// TwinCAT 3 PLC project PlcIotHttpSampleMindsphere
// ProgramVersion: 3.1.4023.0
// libraries:
//   Tc2_Standard, * (Beckhoff Automation GmbH)
//   Tc2_System, * (Beckhoff Automation GmbH)
//   Tc3_IotBase, * (Beckhoff Automation GmbH)
//   Tc3_Module, * (Beckhoff Automation GmbH)
// project tree:
//   / PlcTask.TcTTO
//   POUs/ MAIN.TcPOU
//   POUs/Mindsphere/ FB_TestHTTP_Mindsphere_AcquireAAT.TcPOU, FB_TestHTTP_Mindsphere_CreateDataSource.TcPOU, FB_TestHTTP_Mindsphere_CreateMapping.TcPOU, FB_TestHTTP_Mindsphere_GetDataSource.TcPOU, FB_TestHTTP_Mindsphere_KeyRotation.TcPOU, FB_TestHTTP_Mindsphere_Onboarding.TcPOU
// real-time tasks:
//   TASK PlcTask: cycle T#10ms, priority 20, ADS port 350

CONFIGURATION PlcIotHttpSampleMindsphere
    RESOURCE PLC ON TwinCAT3
        TASK PlcTask(INTERVAL := T#10ms, PRIORITY := 20);
        PROGRAM MAIN WITH PlcTask : MAIN;
    END_RESOURCE
END_CONFIGURATION

// ---- POUs/MAIN.TcPOU
PROGRAM MAIN
VAR
	// trigger command execution for Siemens Mindsphere samples
	bOnboardMindsphere				: BOOL;
	bKeyRotationMindsphere			: BOOL;
	bAcquireAATMindsphere			: BOOL;
	bCreateDataSourceMindsphere		: BOOL;
	bGetDataSourceMindsphere		: BOOL;
	bCreateMappingMindsphere		: BOOL;
	
	fbHttpClientMindsphere			: FB_IotHttpClient :=(sHostName:='gateway.eu1.mindsphere.io',
									bKeepAlive:=TRUE, tConnectionTimeout:=T#10S);						
	
	fbHttpMindsphereOnboarding		: FB_TestHTTP_Mindsphere_Onboarding;
	fbHttpMindsphereKeyRotation		: FB_TestHTTP_Mindsphere_KeyRotation;
	fbHttpMindsphereAcquireAAT		: FB_TestHTTP_Mindsphere_AcquireAAT;
	fbHttpMindsphereCreateDataSource: FB_TestHTTP_Mindsphere_CreateDataSource;
	fbHttpMindsphereGetDataSource	: FB_TestHTTP_Mindsphere_GetDataSource;
	fbHttpMindsphereCreateMapping	: FB_TestHTTP_Mindsphere_CreateMapping;
END_VAR

// init client parameters at startup
IF NOT fbHttpClientMindsphere.bConfigured THEN 
	fbHttpClientMindsphere.stTLS.sCA:= 'C:\TwinCAT\3.1\Config\Certificates\Mindsphere\MindsphereRoot_Europe.pem';
	fbHttpClientMindsphere.nHostPort:= 443;
	fbHttpClientMindsphere.stTLS.bNoServerCertCheck:= TRUE;
END_IF

IF fbHttpClientMindsphere.bConfigured THEN
 	fbHttpMindsphereOnboarding(bSend:=bOnboardMindsphere, fbClient:=fbHttpClientMindsphere);
	fbHttpMindsphereKeyRotation(bSend:=bKeyRotationMindsphere, fbClient:=fbHttpClientMindsphere);
	fbHttpMindsphereAcquireAAT(bSend:=bAcquireAATMindsphere, fbClient:=fbHttpClientMindsphere);
	fbHttpMindsphereCreateDataSource(bSend:=bCreateDataSourceMindsphere, fbClient:=fbHttpClientMindsphere);
	fbHttpMindsphereGetDataSource(bSend:=bGetDataSourceMindsphere, fbClient:=fbHttpClientMindsphere);
	fbHttpMindsphereCreateMapping(bSend:=bCreateMappingMindsphere, fbClient:=fbHttpClientMindsphere);
END_IF

fbHttpClientMindsphere.Execute();

END_PROGRAM

// ---- POUs/Mindsphere/FB_TestHTTP_Mindsphere_Onboarding.TcPOU
FUNCTION_BLOCK FB_TestHTTP_Mindsphere_Onboarding
VAR_INPUT
	bSend				: BOOL;
END_VAR
VAR_IN_OUT
	fbClient			: FB_IotHttpClient;
END_VAR
VAR_OUTPUT
	bBusy				: BOOL;
	bError				: BOOL;
END_VAR
VAR	
	fbRequest			: FB_IotHttpRequest;
	fbHeader			: FB_IotHttpHeaderFieldMap;
	fbJson				: FB_JsonDomParser;
	nState				: UDINT;
	RisingEdge			: R_TRIG;
	
	bGetContentResult	: BOOL;
	sContent			: STRING(2048);
	
	bGetJsonResult		: BOOL;
	jsonDoc				: SJsonValue;
	jsonVal				: SJsonValue;
	sResultValue		: STRING;
	
	nReqCount			: UDINT;
	nResCount			: UDINT;
	nValidResCount		: UDINT;
	nErrCount			: UDINT;	
END_VAR

RisingEdge(CLK:= bSend);
CASE nState OF
0:		
	IF RisingEdge.Q THEN
		sContent := '{}';
		fbHeader.AddField('Content-Type', 'application/json', FALSE);
		fbHeader.AddField('Authorization', 'Bearer eyJraWQiOiJrZXktaWQtMSIsInR5cCI6IkpXVCIsImFsZyI6IlJTMjU2In0.eyJpc3MiOiJTQ0kiLCJzdWIiOiI5NTZjY2UzNjA1YjE0MjA4OTAwOTVlNTBlMmIxMWUxNyIsImF1ZCI6IkFJQU0iLCJpYXQiOjE1ODIxODUxMzMsIm5iZiI6MTU4MjE4NTEzMywiZXhwIjoxNTgyNzg5OTMzLCJqdGkiOiIxYWI0Y2U4MS1jOWJhLTQ2MzctYjIyNy0xYmZjNjk5MWI4NGEiLCJzY29wZSI6IklBVCIsInRlbiI6ImJlY2tob2ZmIiwidGVuX2N0eCI6Im1haW4tdGVuYW50IiwiY2xpZW50X2NyZWRlbnRpYWxzX3Byb2ZpbGUiOlsiU0hBUkVEX1NFQ1JFVCJdLCJzY2hlbWFzIjpbInVybjpzaWVtZW5zOm1pbmRzcGhlcmU6djEiXX0.mOtfZ4WU-8C8r2SggtAEXPS6e1dGlTl4IhrB8WwrWN-FoJE5Tq1DR5j2pSnBRtEuBcrJhd3_Lu2kQ_YdJxJwrPnw_7XdTjqc-LavqDZUUZhOQGqVCurarsKkKcYUMGC8WDLXG81z64l4vrjYSC6drq7ZXVYZVWa-MyHQSWoxQ9QJv1hy_dNYjL6mNf6rmlSqhbzQGo3-3_y5pb7AptIPwYB7GHeH5Iw28PJxjjrWP18ifQlDZYz4AmLGYzdyvGWbbAeHjrdkI8GXls7yhBZ_xIcFwYT72UsDaxG_SIA5YqWhBCyyNM-ElInfPW2PAwe3irzbxinKO3uhstYjJqN3Rg', FALSE);
		IF fbRequest.SendRequest(sUri:= '/api/agentmanagement/v3/register', fbClient:= fbClient, eRequestType:= ETcIotHttpRequestType.HTTP_POST, pContent:= ADR(sContent), nContentSize:= LEN2(ADR(sContent)), fbHeader:= fbHeader) THEN				
			nState:= 1;
			nReqCount:= nReqCount+1;
			bBusy:= TRUE;
			bError:= FALSE;
		END_IF					
	END_IF
1:
	IF NOT fbRequest.bBusy THEN
		bError:= TRUE;
		IF NOT fbRequest.bError THEN				 				
			bGetContentResult:= fbRequest.GetContent(pContent:= ADR(sContent), nContentSize:= SIZEOF(sContent), bSetNullTermination:= TRUE);	
			IF fbRequest.nStatusCode >= 200 AND fbRequest.nStatusCode < 300 THEN
				bGetJsonResult:= FALSE;
				jsonDoc:= fbRequest.GetJsonDomContent(fbJson);				
				(* Parse Onboarding response in order to acquire:
					client_id
					client_secret
					client_secret_expires_at
					regsitration_access_token (RAT)
					registration_client_uri 
				*)
				nResCount:= nResCount+1;					
			END_IF				
		END_IF
		nState:= 0;
		bBusy:= FALSE;
		IF bError THEN
			nErrCount:= nErrCount+1;
		END_IF		
	END_IF  	
END_CASE

END_FUNCTION_BLOCK

// ---- POUs/Mindsphere/FB_TestHTTP_Mindsphere_KeyRotation.TcPOU
FUNCTION_BLOCK FB_TestHTTP_Mindsphere_KeyRotation
VAR_INPUT
	bSend				: BOOL;
END_VAR
VAR_IN_OUT
	fbClient			: FB_IotHttpClient;
END_VAR
VAR_OUTPUT
	bBusy				: BOOL;
	bError				: BOOL;
END_VAR
VAR	
	fbRequest			: FB_IotHttpRequest;
	fbHeader			: FB_IotHttpHeaderFieldMap;
	fbJson				: FB_JsonDomParser;
	nState				: UDINT;
	RisingEdge			: R_TRIG;
	
	bGetContentResult	: BOOL;
	sContent			: STRING(2048);
	
	bGetJsonResult		: BOOL;
	jsonDoc				: SJsonValue;
	jsonVal				: SJsonValue;
	sResultValue		: STRING;
	
	nReqCount			: UDINT;
	nResCount			: UDINT;
	nValidResCount		: UDINT;
	nErrCount			: UDINT;	
END_VAR

RisingEdge(CLK:= bSend);
CASE nState OF
0:		
	IF RisingEdge.Q THEN
		sContent := '{ "client_id": "956cce3605b1420890095e50e2b11e17" }';
		fbHeader.AddField('Content-Type', 'application/json', FALSE);
		// Header field 'Authorization' now includes RAT 
		fbHeader.AddField('Authorization', 'Bearer eyJraWQiOiJrZXktaWQtMSIsInR5cCI6IkpXVCIsImFsZyI6IlJTMjU2In0.eyJpc3MiOiJTQ0kiLCJzdWIiOiI5NTZjY2UzNjA1YjE0MjA4OTAwOTVlNTBlMmIxMWUxNyIsImF1ZCI6IkFJQU0iLCJpYXQiOjE1ODIxODcwNTEsIm5iZiI6MTU4MjE4NzA1MSwiZXhwIjozMTU1Njg4OTg2NDQwMzE5OSwianRpIjoiNzYzM2ViZjctNWY1ZS00NWI3LTkwOTctYzEyODRkZWU2ZjNjIiwic2NvcGUiOiJSQVQiLCJ0ZW4iOiJiZWNraG9mZiIsInRlbl9jdHgiOiJtYWluLXRlbmFudCIsImNsaWVudF9jcmVkZW50aWFsc19wcm9maWxlIjpbIlNIQVJFRF9TRUNSRVQiXSwic2NoZW1hcyI6WyJ1cm46c2llbWVuczptaW5kc3BoZXJlOnYxIl19.dE3IGrI0JIY6O6nYmLp0F3yxHYIvTzQtT9d7ZL7X5MdKMXUeO6G_nXl2MFgEnThPm400hqtsOkLUO1MptoFFlg3rOj227p2--hYN4zLIefDKd54tG0dZ0K7HuX7_oMBjRKoUzF6ls7ujfGyjYH4o0A3FW42mZCecmZxLJmcYoWi7J5iF6oLMZc--Yg1O5RTXwkjp0pwRNMJVS_xofNAdPxg3wvIYjsraUl_TGLPswG_JnsNuYhnRtGfrG23zg1IlSszkB-RYwnzLvsep6ACAfVRlsJve0CN6zU87W0GboH7s_aDAAVTlxbNMz3Tvu44gOk0FmhDoMOvb20peNyg9Iw', FALSE);
		IF fbRequest.SendRequest(sUri:= '/api/agentmanagement/v3/register/956cce3605b1420890095e50e2b11e17', fbClient:= fbClient, eRequestType:= ETcIotHttpRequestType.HTTP_PUT, pContent:= ADR(sContent), nContentSize:= LEN2(ADR(sContent)), fbHeader:= fbHeader) THEN				
			nState:= 1;
			nReqCount:= nReqCount+1;
			bBusy:= TRUE;
			bError:= FALSE;
		END_IF					
	END_IF
1:
	IF NOT fbRequest.bBusy THEN
		bError:= TRUE;
		IF NOT fbRequest.bError THEN				 				
			bGetContentResult:= fbRequest.GetContent(pContent:= ADR(sContent), nContentSize:= SIZEOF(sContent), bSetNullTermination:= TRUE);	
			IF fbRequest.nStatusCode >= 200 AND fbRequest.nStatusCode < 300 THEN
				bGetJsonResult:= FALSE;
				jsonDoc:= fbRequest.GetJsonDomContent(fbJson);				
				(* Parse KeyRotation response in order to acquire:
					client_id
					client_secret
					client_secret_expires_at
					regsitration_access_token (RAT)
					registration_client_uri 
				*)
				nResCount:= nResCount+1;					
			END_IF				
		END_IF
		nState:= 0;
		bBusy:= FALSE;
		IF bError THEN
			nErrCount:= nErrCount+1;
		END_IF		
	END_IF  	
END_CASE

END_FUNCTION_BLOCK

// ---- POUs/Mindsphere/FB_TestHTTP_Mindsphere_AcquireAAT.TcPOU
FUNCTION_BLOCK FB_TestHTTP_Mindsphere_AcquireAAT
VAR_INPUT
	bSend				: BOOL;
END_VAR
VAR_IN_OUT
	fbClient			: FB_IotHttpClient;
END_VAR
VAR_OUTPUT
	bBusy				: BOOL;
	bError				: BOOL;
END_VAR
VAR	
	fbRequest			: FB_IotHttpRequest;
	fbHeader			: FB_IotHttpHeaderFieldMap;
	fbJson				: FB_JsonDomParser;
	nState				: UDINT;
	RisingEdge			: R_TRIG;
	
	bGetContentResult	: BOOL;
	sContent			: STRING(2048);
	
	bGetJsonResult		: BOOL;
	jsonDoc				: SJsonValue;
	jsonVal				: SJsonValue;
	sResultValue		: STRING;
	
	nReqCount			: UDINT;
	nResCount			: UDINT;
	nValidResCount		: UDINT;
	nErrCount			: UDINT;	
END_VAR

RisingEdge(CLK:= bSend);
CASE nState OF
0:		
	IF RisingEdge.Q THEN
		sContent := 'grant_type=client_credentials&client_assertion_type=urn:ietf:params:oauth:client-assertion-type:jwt-bearer&client_assertion=eyJ0eXAiOiJKV1QiLCJhbGciOiJIUzI1NiJ9.eyJpc3MiOiI5NTZjY2UzNjA1YjE0MjA4OTAwOTVlNTBlMmIxMWUxNyIsInN1YiI6Ijk1NmNjZTM2MDViMTQyMDg5MDA5NWU1MGUyYjExZTE3IiwiYXVkIjpbInNvdXRoZ2F0ZSJdLCJpYXQiOjE1ODIxOTI2NjEsIm5iZiI6MTU4MjE5MjY2MSwiZXhwIjoxNTgyMTkzNjYxLCJqdGkiOiJjNDJlYjNiYy04NjI2LTQ3ZDktOTRjYy01MWE0OGQ3ZTc3YjMiLCJ0ZW4iOiJiZWNraG9mZiIsInNjaGVtYXMiOlsidXJuOnNpZW1lbnM6bWluZHNwaGVyZTp2MSJdfQ.LZcYDd38oRX1rdwGeBuqJVy5S4ja4Bmo5lvTW-EloP4';
		fbHeader.AddField('Content-Type', 'application/x-www-form-urlencoded', FALSE);
		IF fbRequest.SendRequest(sUri:= '/api/agentmanagement/v3/oauth/token', fbClient:= fbClient, eRequestType:= ETcIotHttpRequestType.HTTP_POST, pContent:= ADR(sContent), nContentSize:= LEN2(ADR(sContent)), fbHeader:= fbHeader) THEN				
			nState:= 1;
			nReqCount:= nReqCount+1;
			bBusy:= TRUE;
			bError:= FALSE;
		END_IF					
	END_IF
1:
	IF NOT fbRequest.bBusy THEN
		bError:= TRUE;
		IF NOT fbRequest.bError THEN				 				
			bGetContentResult:= fbRequest.GetContent(pContent:= ADR(sContent), nContentSize:= SIZEOF(sContent), bSetNullTermination:= TRUE);	
			IF fbRequest.nStatusCode >= 200 AND fbRequest.nStatusCode < 300 THEN
				bGetJsonResult:= FALSE;
				jsonDoc:= fbRequest.GetJsonDomContent(fbJson);				
				(* Parse AAT API Call response in order to acquire:
					access_token
					token_type
					expires_in
					scope
					jti 
				*)
				nResCount:= nResCount+1;					
			END_IF				
		END_IF
		nState:= 0;
		bBusy:= FALSE;
		IF bError THEN
			nErrCount:= nErrCount+1;
		END_IF		
	END_IF  	
END_CASE

END_FUNCTION_BLOCK

// ---- POUs/Mindsphere/FB_TestHTTP_Mindsphere_CreateDataSource.TcPOU
FUNCTION_BLOCK FB_TestHTTP_Mindsphere_CreateDataSource
VAR_INPUT
	bSend				: BOOL;
END_VAR
VAR_IN_OUT
	fbClient			: FB_IotHttpClient;
END_VAR
VAR_OUTPUT
	bBusy				: BOOL;
	bError				: BOOL;
END_VAR
VAR	
	fbRequest			: FB_IotHttpRequest;
	fbHeader			: FB_IotHttpHeaderFieldMap;
	fbJson				: FB_JsonDomParser;
	nState				: UDINT;
	RisingEdge			: R_TRIG;
	
	bGetContentResult	: BOOL;
	sContent			: STRING(2048);
	
	bGetJsonResult		: BOOL;
	jsonDoc				: SJsonValue;
	jsonVal				: SJsonValue;
	sResultValue		: STRING;
	
	nReqCount			: UDINT;
	nResCount			: UDINT;
	nValidResCount		: UDINT;
	nErrCount			: UDINT;	
END_VAR

RisingEdge(CLK:= bSend);
CASE nState OF
0:		
	IF RisingEdge.Q THEN
		// Body includes JSON document with DataSource configuration that should be created
		sContent := '{"configurationId":"Device_DataSource","dataSources":[{"name":"Device_DataSource_Data","customData":null,"description":"","dataPoints":[{"id":"PWR_OUT","name":"PWR_OUT","description":"","unit":"MW","type":"DOUBLE","customData":null},{"id":"V_OUT","name":"V_OUT","description":"","unit":"Volt","type":"DOUBLE","customData":null}]}]}';
		fbHeader.AddField('Content-Type', 'application/json', FALSE);
		fbHeader.AddField('If-Match', '0', FALSE);
		// Header field 'Authorization' now includes AAT 
		fbHeader.AddField('Authorization', 'Bearer eyJraWQiOiJrZXktaWQtMSIsImFsZyI6IlJTMjU2IiwidHlwIjoiSldUIn0.eyJqdGkiOiJjNzgzOTg1OC1mYmQ4LTQ5YTQtOTE5Yy03YjFmN2FiMDQ3ZjUiLCJzY29wZSI6WyJtZHNwOmNvcmU6RGVmYXVsdEFnZW50Il0sImlzcyI6Imh0dHBzOi8vc291dGhnYXRlLmV1MS5taW5kc3BoZXJlLmlvL2FwaS9hZ2VudG1hbmFnZW1lbnQvIiwic3ViIjoiZTFmODRkM2VkMGIzNDljY2JjYWQxZTkwMzgxMzE5ZTIiLCJ6aWQiOiJhZ2VudGlhbSIsImF1ZCI6WyJzb3V0aGdhdGUiXSwiaWF0IjoxNTgyMTkzMjQ3LCJleHAiOjE1ODIxOTY4NDcsInNjaGVtYXMiOlsidXJuOnNpZW1lbnM6bWluZHNwaGVyZTppYW06djEiXSwidGVuIjoiYmVja2hvZmYiLCJ0ZW5fY3R4IjoibWFpbi10ZW5hbnQiLCJjYXQiOiJhZ2VudC10b2tlbjp2MSIsImdyYW50X3R5cGUiOiJjbGllbnRfY3JlZGVudGlhbHMifQ.IAg9zGZaXy-qHVr5SVTFePF8mnZQjG6uwEIXtmsESyFrdhkJJTa3rnaksMMAvr9mPyXelYhvnw0GcWhQtCRFDfKFV5jTXfXsRaSNFPO_2Um6H37JFt6coWqmO6woiKkFKHTw3CiuUEc-Rl0XgzEXQThbDQCeQzaD3jcog44Nmp8R2rm4BoDzeQk2wsvpEPJeZEzCTFLdfWxodmQT7yHA0P_UMC58ztSB2FlM3NTUl_NhEFF3unf5DgIRe8nTQhY8eH09r9Ni0PiqQTbhsxWQg3mB-bOM1imlgnveO5vRlcZi96-HM78DtDM3HpZdgTOLny1jykSv0JHwe-UD7bvqww', FALSE);
		IF fbRequest.SendRequest(sUri:= '/api/agentmanagement/v3/agents/e1f84d3ed0b349ccbcad1e90381319e2/dataSourceConfiguration', fbClient:= fbClient, eRequestType:= ETcIotHttpRequestType.HTTP_PUT, pContent:= ADR(sContent), nContentSize:= LEN2(ADR(sContent)), fbHeader:= fbHeader) THEN				
			nState:= 1;
			nReqCount:= nReqCount+1;
			bBusy:= TRUE;
			bError:= FALSE;
		END_IF					
	END_IF
1:
	IF NOT fbRequest.bBusy THEN
		bError:= TRUE;
		IF NOT fbRequest.bError THEN				 				
			bGetContentResult:= fbRequest.GetContent(pContent:= ADR(sContent), nContentSize:= SIZEOF(sContent), bSetNullTermination:= TRUE);	
			IF fbRequest.nStatusCode >= 200 AND fbRequest.nStatusCode < 300 THEN
				bGetJsonResult:= FALSE;
				jsonDoc:= fbRequest.GetJsonDomContent(fbJson);				
				(* Parse response in order to acquire created DatsSource configuration *)
				nResCount:= nResCount+1;					
			END_IF				
		END_IF
		nState:= 0;
		bBusy:= FALSE;
		IF bError THEN
			nErrCount:= nErrCount+1;
		END_IF		
	END_IF  	
END_CASE

END_FUNCTION_BLOCK

// ---- POUs/Mindsphere/FB_TestHTTP_Mindsphere_GetDataSource.TcPOU
FUNCTION_BLOCK FB_TestHTTP_Mindsphere_GetDataSource
VAR_INPUT
	bSend				: BOOL;
END_VAR
VAR_IN_OUT
	fbClient			: FB_IotHttpClient;
END_VAR
VAR_OUTPUT
	bBusy				: BOOL;
	bError				: BOOL;
END_VAR
VAR	
	fbRequest			: FB_IotHttpRequest;
	fbHeader			: FB_IotHttpHeaderFieldMap;
	fbJson				: FB_JsonDomParser;
	nState				: UDINT;
	RisingEdge			: R_TRIG;
	
	bGetContentResult	: BOOL;
	sContent			: STRING(2048);
	
	bGetJsonResult		: BOOL;
	jsonDoc				: SJsonValue;
	jsonVal				: SJsonValue;
	sResultValue		: STRING;
	
	nReqCount			: UDINT;
	nResCount			: UDINT;
	nValidResCount		: UDINT;
	nErrCount			: UDINT;	
END_VAR

RisingEdge(CLK:= bSend);
CASE nState OF
0:		
	IF RisingEdge.Q THEN
		sContent := '';
		fbHeader.AddField('Content-Type', 'application/x-www-form-urlencoded', FALSE);
		// Header field 'Authorization' now includes RAT 
		fbHeader.AddField('Authorization', 'Bearer eyJraWQiOiJrZXktaWQtMSIsImFsZyI6IlJTMjU2IiwidHlwIjoiSldUIn0.eyJqdGkiOiJlY2I4Y2RkZS1jOTFhLTRkNGMtODA2Mi1lYTBmN2Y5ZGZkMjkiLCJzY29wZSI6WyJtZHNwOmNvcmU6RGVmYXVsdEFnZW50Il0sImlzcyI6Imh0dHBzOi8vc291dGhnYXRlLmV1MS5taW5kc3BoZXJlLmlvL2FwaS9hZ2VudG1hbmFnZW1lbnQvIiwic3ViIjoiOTU2Y2NlMzYwNWIxNDIwODkwMDk1ZTUwZTJiMTFlMTciLCJ6aWQiOiJhZ2VudGlhbSIsImF1ZCI6WyJzb3V0aGdhdGUiXSwiaWF0IjoxNTgyMTg4OTIwLCJleHAiOjE1ODIxOTI1MjAsInNjaGVtYXMiOlsidXJuOnNpZW1lbnM6bWluZHNwaGVyZTppYW06djEiXSwidGVuIjoiYmVja2hvZmYiLCJ0ZW5fY3R4IjoibWFpbi10ZW5hbnQiLCJjYXQiOiJhZ2VudC10b2tlbjp2MSIsImdyYW50X3R5cGUiOiJjbGllbnRfY3JlZGVudGlhbHMifQ.XLMR7pQDBiRZeDwtBLfKujJrPIWwvFw28DjtedfYL_x4iOUIcV7U6AJyKe6Wnit4GOAKfJYh_BGD160E3ns7RjRBYSx8Lj5dxI20l3g_KMcpgILoaW8gYlx41Y4q6W44zctJ04TQLsaz-Vc3eOEJ_TdMTGc_7s4v4YsQbZinKN-ZmQF_sXdGbihL2CkbqhnaubwZGn_FmSZosuiDXk4GFdF1TX2xXHQCz39p8jPYtgq2x9LkuIFtEzUct_lTy30rcwS2Fq6m-ac6gldJFtvqLZoXu3wUlHR1F7kAYndm6wvtXXlgDo5otTMZfzXBTEQA3JS2Cucys3gJNhYEDpUAtg', FALSE);
		IF fbRequest.SendRequest(sUri:= '/api/agentmanagement/v3/agents/956cce3605b1420890095e50e2b11e17/dataSourceConfiguration', fbClient:= fbClient, eRequestType:= ETcIotHttpRequestType.HTTP_GET, pContent:= ADR(sContent), nContentSize:= LEN2(ADR(sContent)), fbHeader:= fbHeader) THEN				
			nState:= 1;
			nReqCount:= nReqCount+1;
			bBusy:= TRUE;
			bError:= FALSE;
		END_IF					
	END_IF
1:
	IF NOT fbRequest.bBusy THEN
		bError:= TRUE;
		IF NOT fbRequest.bError THEN				 				
			bGetContentResult:= fbRequest.GetContent(pContent:= ADR(sContent), nContentSize:= SIZEOF(sContent), bSetNullTermination:= TRUE);	
			IF fbRequest.nStatusCode >= 200 AND fbRequest.nStatusCode < 300 THEN
				bGetJsonResult:= FALSE;
				jsonDoc:= fbRequest.GetJsonDomContent(fbJson);				
				(* Parse response in order to acquire DataSource configuration for this asset *)
				nResCount:= nResCount+1;					
			END_IF				
		END_IF
		nState:= 0;
		bBusy:= FALSE;
		IF bError THEN
			nErrCount:= nErrCount+1;
		END_IF		
	END_IF  	
END_CASE

END_FUNCTION_BLOCK

// ---- POUs/Mindsphere/FB_TestHTTP_Mindsphere_CreateMapping.TcPOU
FUNCTION_BLOCK FB_TestHTTP_Mindsphere_CreateMapping
VAR_INPUT
	bSend				: BOOL;
END_VAR
VAR_IN_OUT
	fbClient			: FB_IotHttpClient;
END_VAR
VAR_OUTPUT
	bBusy				: BOOL;
	bError				: BOOL;
END_VAR
VAR	
	fbRequest			: FB_IotHttpRequest;
	fbHeader			: FB_IotHttpHeaderFieldMap;
	fbJson				: FB_JsonDomParser;
	nState				: UDINT;
	RisingEdge			: R_TRIG;
	
	bGetContentResult	: BOOL;
	sContent			: STRING(2048);
	
	bGetJsonResult		: BOOL;
	jsonDoc				: SJsonValue;
	jsonVal				: SJsonValue;
	sResultValue		: STRING;
	
	nReqCount			: UDINT;
	nResCount			: UDINT;
	nValidResCount		: UDINT;
	nErrCount			: UDINT;	
END_VAR

RisingEdge(CLK:= bSend);
CASE nState OF
0:		
	IF RisingEdge.Q THEN
		// Body includes JSON document with DataSource configuration that should be created
		sContent := '{"agentId":"956cce3605b1420890095e50e2b11e17","dataPointId":"DP001_temprature_KLR","entityId":"956cce3605b1420890095e50e2b11e17","propertySetName":"SvenG_NB05_Aspect","propertyName":"Pump1"}';
		fbHeader.AddField('Content-Type', 'application/json', FALSE);
		// Header field 'Authorization' now includes RAT 
		fbHeader.AddField('Authorization', 'Bearer eyJraWQiOiJrZXktaWQtMSIsImFsZyI6IlJTMjU2IiwidHlwIjoiSldUIn0.eyJqdGkiOiJlY2I4Y2RkZS1jOTFhLTRkNGMtODA2Mi1lYTBmN2Y5ZGZkMjkiLCJzY29wZSI6WyJtZHNwOmNvcmU6RGVmYXVsdEFnZW50Il0sImlzcyI6Imh0dHBzOi8vc291dGhnYXRlLmV1MS5taW5kc3BoZXJlLmlvL2FwaS9hZ2VudG1hbmFnZW1lbnQvIiwic3ViIjoiOTU2Y2NlMzYwNWIxNDIwODkwMDk1ZTUwZTJiMTFlMTciLCJ6aWQiOiJhZ2VudGlhbSIsImF1ZCI6WyJzb3V0aGdhdGUiXSwiaWF0IjoxNTgyMTg4OTIwLCJleHAiOjE1ODIxOTI1MjAsInNjaGVtYXMiOlsidXJuOnNpZW1lbnM6bWluZHNwaGVyZTppYW06djEiXSwidGVuIjoiYmVja2hvZmYiLCJ0ZW5fY3R4IjoibWFpbi10ZW5hbnQiLCJjYXQiOiJhZ2VudC10b2tlbjp2MSIsImdyYW50X3R5cGUiOiJjbGllbnRfY3JlZGVudGlhbHMifQ.XLMR7pQDBiRZeDwtBLfKujJrPIWwvFw28DjtedfYL_x4iOUIcV7U6AJyKe6Wnit4GOAKfJYh_BGD160E3ns7RjRBYSx8Lj5dxI20l3g_KMcpgILoaW8gYlx41Y4q6W44zctJ04TQLsaz-Vc3eOEJ_TdMTGc_7s4v4YsQbZinKN-ZmQF_sXdGbihL2CkbqhnaubwZGn_FmSZosuiDXk4GFdF1TX2xXHQCz39p8jPYtgq2x9LkuIFtEzUct_lTy30rcwS2Fq6m-ac6gldJFtvqLZoXu3wUlHR1F7kAYndm6wvtXXlgDo5otTMZfzXBTEQA3JS2Cucys3gJNhYEDpUAtg', FALSE);
		IF fbRequest.SendRequest(sUri:= '/api/mindconnect/v3/dataPointMappings', fbClient:= fbClient, eRequestType:= ETcIotHttpRequestType.HTTP_POST, pContent:= ADR(sContent), nContentSize:= LEN2(ADR(sContent)), fbHeader:= fbHeader) THEN				
			nState:= 1;
			nReqCount:= nReqCount+1;
			bBusy:= TRUE;
			bError:= FALSE;
		END_IF					
	END_IF
1:
	IF NOT fbRequest.bBusy THEN
		bError:= TRUE;
		IF NOT fbRequest.bError THEN				 				
			bGetContentResult:= fbRequest.GetContent(pContent:= ADR(sContent), nContentSize:= SIZEOF(sContent), bSetNullTermination:= TRUE);	
			IF fbRequest.nStatusCode >= 200 AND fbRequest.nStatusCode < 300 THEN
				bGetJsonResult:= FALSE;
				jsonDoc:= fbRequest.GetJsonDomContent(fbJson);				
				(* Parse response in order to acquire created DatsSource configuration *)
				nResCount:= nResCount+1;					
			END_IF				
		END_IF
		nState:= 0;
		bBusy:= FALSE;
		IF bError THEN
			nErrCount:= nErrCount+1;
		END_IF		
	END_IF  	
END_CASE

END_FUNCTION_BLOCK
